    stLENS1_750[835].fEnergy := 31673.702636; stLENS1_750[835].fLow := 3.913613; stLENS1_750[835].fHigh := 9.337805; 
    stLENS1_750[836].fEnergy := 31737.113431; stLENS1_750[836].fLow := 3.899151; stLENS1_750[836].fHigh := 9.298086; 
    stLENS1_750[837].fEnergy := 31800.651174; stLENS1_750[837].fLow := 3.884743; stLENS1_750[837].fHigh := 9.258535; 
    stLENS1_750[838].fEnergy := 31864.316120; stLENS1_750[838].fLow := 3.870389; stLENS1_750[838].fHigh := 9.219153; 
    stLENS1_750[839].fEnergy := 31928.108524; stLENS1_750[839].fLow := 3.856087; stLENS1_750[839].fHigh := 9.179939; 
    stLENS1_750[840].fEnergy := 31992.028640; stLENS1_750[840].fLow := 3.841838; stLENS1_750[840].fHigh := 9.140891; 
    stLENS1_750[841].fEnergy := 32056.076724; stLENS1_750[841].fLow := 3.827642; stLENS1_750[841].fHigh := 9.102009; 
    stLENS1_750[842].fEnergy := 32120.253032; stLENS1_750[842].fLow := 3.813498; stLENS1_750[842].fHigh := 9.063293; 
    stLENS1_750[843].fEnergy := 32184.557822; stLENS1_750[843].fLow := 3.799407; stLENS1_750[843].fHigh := 9.024741; 
    stLENS1_750[844].fEnergy := 32248.991349; stLENS1_750[844].fLow := 3.785367; stLENS1_750[844].fHigh := 8.986354; 
    stLENS1_750[845].fEnergy := 32313.553873; stLENS1_750[845].fLow := 3.771380; stLENS1_750[845].fHigh := 8.948129; 
    stLENS1_750[846].fEnergy := 32378.245651; stLENS1_750[846].fLow := 3.757444; stLENS1_750[846].fHigh := 8.910067; 
    stLENS1_750[847].fEnergy := 32443.066942; stLENS1_750[847].fLow := 3.743559; stLENS1_750[847].fHigh := 8.872167; 
    stLENS1_750[848].fEnergy := 32508.018005; stLENS1_750[848].fLow := 3.729726; stLENS1_750[848].fHigh := 8.834429; 
    stLENS1_750[849].fEnergy := 32573.099101; stLENS1_750[849].fLow := 3.715944; stLENS1_750[849].fHigh := 8.796851; 
    stLENS1_750[850].fEnergy := 32638.310488; stLENS1_750[850].fLow := 3.702213; stLENS1_750[850].fHigh := 8.759432; 
    stLENS1_750[851].fEnergy := 32703.652430; stLENS1_750[851].fLow := 3.688533; stLENS1_750[851].fHigh := 8.722173; 
    stLENS1_750[852].fEnergy := 32769.125185; stLENS1_750[852].fLow := 3.674903; stLENS1_750[852].fHigh := 8.685073; 
    stLENS1_750[853].fEnergy := 32834.729018; stLENS1_750[853].fLow := 3.661324; stLENS1_750[853].fHigh := 8.648130; 
    stLENS1_750[854].fEnergy := 32900.464189; stLENS1_750[854].fLow := 3.647795; stLENS1_750[854].fHigh := 8.611344; 
    stLENS1_750[855].fEnergy := 32966.330962; stLENS1_750[855].fLow := 3.634316; stLENS1_750[855].fHigh := 8.574715; 
    stLENS1_750[856].fEnergy := 33032.329601; stLENS1_750[856].fLow := 3.620886; stLENS1_750[856].fHigh := 8.538241; 
    stLENS1_750[857].fEnergy := 33098.460369; stLENS1_750[857].fLow := 3.607507; stLENS1_750[857].fHigh := 8.501923; 
    stLENS1_750[858].fEnergy := 33164.723530; stLENS1_750[858].fLow := 3.594176; stLENS1_750[858].fHigh := 8.465759; 
    stLENS1_750[859].fEnergy := 33231.119351; stLENS1_750[859].fLow := 3.580895; stLENS1_750[859].fHigh := 8.429749; 
    stLENS1_750[860].fEnergy := 33297.648096; stLENS1_750[860].fLow := 3.567663; stLENS1_750[860].fHigh := 8.393893; 
    stLENS1_750[861].fEnergy := 33364.310032; stLENS1_750[861].fLow := 3.554480; stLENS1_750[861].fHigh := 8.358188; 
    stLENS1_750[862].fEnergy := 33431.105426; stLENS1_750[862].fLow := 3.541346; stLENS1_750[862].fHigh := 8.322636; 
    stLENS1_750[863].fEnergy := 33498.034543; stLENS1_750[863].fLow := 3.528260; stLENS1_750[863].fHigh := 8.287235; 
    stLENS1_750[864].fEnergy := 33565.097653; stLENS1_750[864].fLow := 3.515222; stLENS1_750[864].fHigh := 8.251984; 
    stLENS1_750[865].fEnergy := 33632.295023; stLENS1_750[865].fLow := 3.502233; stLENS1_750[865].fHigh := 8.216883; 
    stLENS1_750[866].fEnergy := 33699.626923; stLENS1_750[866].fLow := 3.489292; stLENS1_750[866].fHigh := 8.181932; 
    stLENS1_750[867].fEnergy := 33767.093621; stLENS1_750[867].fLow := 3.476398; stLENS1_750[867].fHigh := 8.147129; 
    stLENS1_750[868].fEnergy := 33834.695387; stLENS1_750[868].fLow := 3.463552; stLENS1_750[868].fHigh := 8.112475; 
    stLENS1_750[869].fEnergy := 33902.432493; stLENS1_750[869].fLow := 3.450754; stLENS1_750[869].fHigh := 8.077968; 
    stLENS1_750[870].fEnergy := 33970.305208; stLENS1_750[870].fLow := 3.438003; stLENS1_750[870].fHigh := 8.043607; 
    stLENS1_750[871].fEnergy := 34038.313804; stLENS1_750[871].fLow := 3.425299; stLENS1_750[871].fHigh := 8.009393; 
    stLENS1_750[872].fEnergy := 34106.458554; stLENS1_750[872].fLow := 3.412642; stLENS1_750[872].fHigh := 7.975324; 
    stLENS1_750[873].fEnergy := 34174.739729; stLENS1_750[873].fLow := 3.400032; stLENS1_750[873].fHigh := 7.941400; 
    stLENS1_750[874].fEnergy := 34243.157604; stLENS1_750[874].fLow := 3.387468; stLENS1_750[874].fHigh := 7.907621; 
    stLENS1_750[875].fEnergy := 34311.712451; stLENS1_750[875].fLow := 3.374951; stLENS1_750[875].fHigh := 7.873985; 
    stLENS1_750[876].fEnergy := 34380.404545; stLENS1_750[876].fLow := 3.362480; stLENS1_750[876].fHigh := 7.840492; 
    stLENS1_750[877].fEnergy := 34449.234161; stLENS1_750[877].fLow := 3.350055; stLENS1_750[877].fHigh := 7.807142; 
    stLENS1_750[878].fEnergy := 34518.201574; stLENS1_750[878].fLow := 3.337676; stLENS1_750[878].fHigh := 7.773933; 
    stLENS1_750[879].fEnergy := 34587.307059; stLENS1_750[879].fLow := 3.325342; stLENS1_750[879].fHigh := 7.740866; 
    stLENS1_750[880].fEnergy := 34656.550894; stLENS1_750[880].fLow := 3.313055; stLENS1_750[880].fHigh := 7.707939; 
    stLENS1_750[881].fEnergy := 34725.933355; stLENS1_750[881].fLow := 3.300813; stLENS1_750[881].fHigh := 7.675153; 
    stLENS1_750[882].fEnergy := 34795.454720; stLENS1_750[882].fLow := 3.288615; stLENS1_750[882].fHigh := 7.642506; 
    stLENS1_750[883].fEnergy := 34865.115267; stLENS1_750[883].fLow := 3.276463; stLENS1_750[883].fHigh := 7.609998; 
    stLENS1_750[884].fEnergy := 34934.915274; stLENS1_750[884].fLow := 3.264356; stLENS1_750[884].fHigh := 7.577628; 
    stLENS1_750[885].fEnergy := 35004.855021; stLENS1_750[885].fLow := 3.252294; stLENS1_750[885].fHigh := 7.545396; 
    stLENS1_750[886].fEnergy := 35074.934788; stLENS1_750[886].fLow := 3.240276; stLENS1_750[886].fHigh := 7.513300; 
    stLENS1_750[887].fEnergy := 35145.154854; stLENS1_750[887].fLow := 3.228303; stLENS1_750[887].fHigh := 7.481342; 
    stLENS1_750[888].fEnergy := 35215.515501; stLENS1_750[888].fLow := 3.216374; stLENS1_750[888].fHigh := 7.449519; 
    stLENS1_750[889].fEnergy := 35286.017010; stLENS1_750[889].fLow := 3.204489; stLENS1_750[889].fHigh := 7.417832; 
    stLENS1_750[890].fEnergy := 35356.659663; stLENS1_750[890].fLow := 3.192648; stLENS1_750[890].fHigh := 7.386279; 
    stLENS1_750[891].fEnergy := 35427.443743; stLENS1_750[891].fLow := 3.180850; stLENS1_750[891].fHigh := 7.354861; 
    stLENS1_750[892].fEnergy := 35498.369532; stLENS1_750[892].fLow := 3.169097; stLENS1_750[892].fHigh := 7.323576; 
    stLENS1_750[893].fEnergy := 35569.437315; stLENS1_750[893].fLow := 3.157386; stLENS1_750[893].fHigh := 7.292425; 
    stLENS1_750[894].fEnergy := 35640.647376; stLENS1_750[894].fLow := 3.145719; stLENS1_750[894].fHigh := 7.261406; 
    stLENS1_750[895].fEnergy := 35712.000000; stLENS1_750[895].fLow := 3.134095; stLENS1_750[895].fHigh := 7.230519; 
    stLENS1_750[896].fEnergy := 35783.495472; stLENS1_750[896].fLow := 3.122514; stLENS1_750[896].fHigh := 7.199763; 
    stLENS1_750[897].fEnergy := 35855.134077; stLENS1_750[897].fLow := 3.110976; stLENS1_750[897].fHigh := 7.169138; 
    stLENS1_750[898].fEnergy := 35926.916104; stLENS1_750[898].fLow := 3.099481; stLENS1_750[898].fHigh := 7.138643; 

    bInitialized := TRUE;
END_IF

END_FUNCTION_BLOCK

// ---- POUs/FB_LENS_SYSTEM.TcPOU
FUNCTION_BLOCK FB_LENS_SYSTEM
VAR_INPUT
    LENSES : ARRAY[1..10] OF LENS;  //Array of lens structures
    COUNT  : INT;                   //Number of lenses
    IF_NONE : LREAL := 10000.0;	    //Effective radius if no lenses are inserted (instead of infinity)
END_VAR
VAR_OUTPUT
    UNKNOWN_FAULT : BOOL;         //Fault for unknown lens state
    EFF_RADII     : REAL; //Calculated effective radii
    IN_COUNT 	  : INT;
END_VAR
VAR
    INDEX : INT;                  //Increment for loop
    KNOWN : INT;                  //Number of known lenses
    RADII : ARRAY[1..10] OF REAL; //Inserted Radii
END_VAR

(* FB_LENS_SYSTEM

Monitor an array of lens objects, updating the effective radius and positions of each.
Both the position of the lenses and the combined radius can cause a fault which is
communicated to the MPS system.

*)

//Check positions of lenses
///////////////////////////
KNOWN := 0; //Tally of known lenses
IN_COUNT := 0;

FOR INDEX := 1 TO COUNT BY 1 DO
    IF LENSES[INDEX].IN THEN
        //Inserted lenses are inserted into array
        RADII[INDEX] := LENSES[INDEX].RADIUS;
        IN_COUNT := IN_COUNT + 1;
    ELSE
        //Removed lenses are set to 0.0
        RADII[INDEX] := 0.0;
    END_IF

    // Count all known lenses
    IF LENSES[INDEX].KNOWN THEN
        KNOWN := KNOWN +1;
    END_IF
END_FOR;

// Make sure we have accounted for all lenses
UNKNOWN_FAULT := NOT (COUNT=KNOWN);

// Calculate effective radii of inserted lens
//////////////////////////////////////////////
EFF_RADII := F_EFF_RADIUS(RADII:=RADII, COUNT:=COUNT, IF_NONE:=LREAL_TO_REAL(IF_NONE));

END_FUNCTION_BLOCK

// ---- POUs/F_EFF_RADIUS.TcPOU
FUNCTION F_EFF_RADIUS : REAL
VAR_INPUT
    RADII : ARRAY[1..10] OF REAL; // Array of Effective Radii
    COUNT : INT;                 //  Number of Lenses
    IF_NONE: REAL;              //  Radius to report if none inserted (-> infinity)
END_VAR
VAR
    INDEX: INT; //Counter for Loop
END_VAR

(*F_EFF_RADIUS

Calculate the effective radius of an array of given lens radii. Non-zero elements
up to the count value are summed in reciprocal space and then inverted to give the
final calculation.
*)

// Initialize
F_EFF_RADIUS := 0.0;

//Sum Reciprocals
WHILE INDEX < COUNT+1 DO
    //Add non-zero element to total
    IF RADII[INDEX] > 0.0 THEN
        F_EFF_RADIUS := F_EFF_RADIUS + 1/RADII[INDEX];
    END_IF
    //Increment
    INDEX := INDEX + 1;
END_WHILE

//Invert if non-zero
/////////////////////
IF F_EFF_RADIUS > 0.0 THEN
    F_EFF_RADIUS := 1/F_EFF_RADIUS;
ELSE
    // B
    F_EFF_RADIUS := IF_NONE;
END_IF

END_FUNCTION

// ---- POUs/Modbus/p_ModbusTx_OutputCoils.TcPOU
PROGRAM p_ModbusTx_OutputCoils
VAR
END_VAR

mb_Output_Coils[0]:=FALSE;  //System Controls
mb_Output_Coils[1]:=FALSE;  //System Controls
mb_Output_Coils[2]:=FALSE;  //System Controls
mb_Output_Coils[3]:=FALSE;  //System Controls
mb_Output_Coils[4]:=FALSE;  //System Controls
mb_Output_Coils[5]:=FALSE;  //System Controls
mb_Output_Coils[6]:=FALSE;  //System Controls
mb_Output_Coils[7]:=FALSE;  //System Controls
mb_Output_Coils[8]:=FALSE;  //System Controls
mb_Output_Coils[9]:=FALSE;  //System Controls
mb_Output_Coils[10]:=FALSE;  //Valve switch controls
mb_Output_Coils[11]:=FALSE;  //Valve switch controls
mb_Output_Coils[12]:=FALSE;  //Valve switch controls
mb_Output_Coils[13]:=FALSE;  //Valve switch controls
mb_Output_Coils[14]:=FALSE;  //Valve switch controls
mb_Output_Coils[15]:=FALSE;  //Valve switch controls
mb_Output_Coils[16]:=FALSE;  //Valve switch controls
mb_Output_Coils[17]:=FALSE;  //Valve switch controls
mb_Output_Coils[18]:=FALSE;  //Valve switch controls
mb_Output_Coils[19]:=FALSE;  //Valve switch controls
mb_Output_Coils[20]:=FALSE;  //Valve switch controls
mb_Output_Coils[21]:=FALSE;  //Valve switch controls
mb_Output_Coils[22]:=FALSE;  //Valve switch controls
mb_Output_Coils[23]:=FALSE;  //Valve switch controls
mb_Output_Coils[24]:=FALSE;  //Valve switch controls
mb_Output_Coils[25]:=FALSE;  //Valve switch controls
mb_Output_Coils[26]:=FALSE;  //Valve switch controls
mb_Output_Coils[27]:=FALSE;  //Valve switch controls
mb_Output_Coils[28]:=FALSE;  //Valve switch controls
mb_Output_Coils[29]:=FALSE;  //Valve switch controls
mb_Output_Coils[30]:=FALSE;  //Valve switch controls
mb_Output_Coils[31]:=FALSE;  //Valve switch controls
mb_Output_Coils[32]:=FALSE;  //Valve switch controls
mb_Output_Coils[33]:=FALSE;  //Valve switch controls
mb_Output_Coils[34]:=FALSE;  //Valve switch controls
mb_Output_Coils[35]:=FALSE;  //Valve switch controls
mb_Output_Coils[36]:=FALSE;  //Valve switch controls
mb_Output_Coils[37]:=FALSE;  //Valve switch controls
mb_Output_Coils[38]:=FALSE;  //Valve switch controls
mb_Output_Coils[39]:=FALSE;  //Valve switch controls
mb_Output_Coils[40]:=FALSE;  //Valve switch controls
mb_Output_Coils[41]:=FALSE;  //Valve switch controls
mb_Output_Coils[42]:=FALSE;  //Valve switch controls
mb_Output_Coils[43]:=FALSE;  //Valve switch controls
mb_Output_Coils[44]:=FALSE;  //Valve switch controls
mb_Output_Coils[45]:=FALSE;  //Valve switch controls
mb_Output_Coils[46]:=FALSE;  //Valve switch controls
mb_Output_Coils[47]:=FALSE;  //Valve switch controls
mb_Output_Coils[48]:=FALSE;  //Valve switch controls
mb_Output_Coils[49]:=FALSE;  //Valve switch controls
mb_Output_Coils[50]:=FALSE;  //Valve switch controls
mb_Output_Coils[51]:=FALSE;  //Valve switch controls
mb_Output_Coils[52]:=FALSE;  //Valve switch controls
mb_Output_Coils[53]:=FALSE;  //Valve switch controls
mb_Output_Coils[54]:=FALSE;  //Valve switch controls
mb_Output_Coils[55]:=FALSE;  //Valve switch controls
mb_Output_Coils[56]:=FALSE;  //Valve switch controls
mb_Output_Coils[57]:=FALSE;  //Valve switch controls
mb_Output_Coils[58]:=FALSE;  //Valve switch controls
mb_Output_Coils[59]:=FALSE;  //Valve switch controls
mb_Output_Coils[60]:=FALSE;  //Valve switch controls
mb_Output_Coils[61]:=FALSE;  //Valve switch controls
mb_Output_Coils[62]:=FALSE;  //Valve switch controls
mb_Output_Coils[63]:=FALSE;  //Valve switch controls
mb_Output_Coils[64]:=FALSE;  //Valve switch controls
mb_Output_Coils[65]:=FALSE;  //Valve switch controls
mb_Output_Coils[66]:=FALSE;  //Valve switch controls
mb_Output_Coils[67]:=FALSE;  //Valve switch controls
mb_Output_Coils[68]:=FALSE;  //Valve switch controls
mb_Output_Coils[69]:=FALSE;  //Valve switch controls
mb_Output_Coils[70]:=FALSE;  //Turbo Controls
mb_Output_Coils[71]:=FALSE;  //Turbo Controls
mb_Output_Coils[72]:=FALSE;  //Turbo Controls
mb_Output_Coils[74]:=FALSE;  //Turbo Controls
mb_Output_Coils[75]:=FALSE;  //Turbo Controls
mb_Output_Coils[76]:=FALSE;  //Turbo Controls
mb_Output_Coils[77]:=FALSE;  //Turbo Controls
mb_Output_Coils[78]:=FALSE;  //Turbo Controls
mb_Output_Coils[79]:=FALSE;  //Turbo Controls
mb_Output_Coils[80]:=FALSE;  //Turbo Controls
mb_Output_Coils[81]:=FALSE;  //Turbo Controls
mb_Output_Coils[82]:=FALSE;  //Turbo Controls
mb_Output_Coils[83]:=FALSE;  //Turbo Controls
mb_Output_Coils[84]:=FALSE;  //Turbo Controls
mb_Output_Coils[85]:=FALSE;  //Turbo Controls
mb_Output_Coils[86]:=FALSE;  //Turbo Controls
mb_Output_Coils[87]:=FALSE;  //Turbo Controls
mb_Output_Coils[88]:=FALSE;  //Turbo Controls
mb_Output_Coils[89]:=FALSE;  //Turbo Controls
mb_Output_Coils[90]:=FALSE;  //Turbo Controls
mb_Output_Coils[91]:=FALSE;  //Turbo Controls
mb_Output_Coils[92]:=FALSE;  //Turbo Controls
mb_Output_Coils[93]:=FALSE;  //Turbo Controls
mb_Output_Coils[94]:=FALSE;  //Turbo Controls
mb_Output_Coils[95]:=FALSE;  //Turbo Controls
mb_Output_Coils[96]:=FALSE;  //Turbo Controls
mb_Output_Coils[97]:=FALSE;  //Turbo Controls
mb_Output_Coils[98]:=FALSE;  //Turbo Controls
mb_Output_Coils[99]:=FALSE;  //Turbo Controls
mb_Output_Coils[100]:=FALSE;  //Turbo Controls
mb_Output_Coils[101]:=FALSE;  //Turbo Controls
mb_Output_Coils[102]:=FALSE;  //Turbo Controls
mb_Output_Coils[103]:=FALSE;  //Turbo Controls
mb_Output_Coils[104]:=FALSE;  //Turbo Controls
mb_Output_Coils[105]:=FALSE;  //Turbo Controls
mb_Output_Coils[106]:=FALSE;  //Turbo Controls
mb_Output_Coils[107]:=FALSE;  //Turbo Controls
mb_Output_Coils[108]:=FALSE;  //Turbo Controls
mb_Output_Coils[109]:=FALSE;  //Turbo Controls
mb_Output_Coils[110]:=FALSE;  //Turbo Controls
mb_Output_Coils[111]:=FALSE;  //Turbo Controls
mb_Output_Coils[112]:=FALSE;  //Turbo Controls
mb_Output_Coils[113]:=FALSE;  //Turbo Controls
mb_Output_Coils[114]:=FALSE;  //Turbo Controls
mb_Output_Coils[115]:=FALSE;  //Turbo Controls
mb_Output_Coils[116]:=FALSE;  //Turbo Controls
mb_Output_Coils[117]:=FALSE;  //Turbo Controls
mb_Output_Coils[118]:=FALSE;  //Turbo Controls
mb_Output_Coils[119]:=FALSE;  //Turbo Controls
//mb_Output_Coils[120]:=vgMXT_GCC_06.xHV_SW;  //CC HV Enable
mb_Output_Coils[121]:=FALSE;  //CC HV Enable
mb_Output_Coils[122]:=FALSE;  //CC HV Enable
mb_Output_Coils[123]:=FALSE;  //CC HV Enable
mb_Output_Coils[124]:=FALSE;  //CC HV Enable
mb_Output_Coils[125]:=FALSE;  //CC HV Enable
mb_Output_Coils[126]:=FALSE;  //CC HV Enable
mb_Output_Coils[127]:=FALSE;  //CC HV Enable
mb_Output_Coils[128]:=FALSE;  //CC HV Enable
mb_Output_Coils[129]:=FALSE;  //CC HV Enable
mb_Output_Coils[130]:=FALSE;  //CC HV Enable
mb_Output_Coils[131]:=FALSE;  //CC HV Enable
mb_Output_Coils[132]:=FALSE;  //CC HV Enable
mb_Output_Coils[133]:=FALSE;  //CC HV Enable
mb_Output_Coils[134]:=FALSE;  //CC HV Enable
mb_Output_Coils[135]:=FALSE;  //CC HV Enable
mb_Output_Coils[136]:=FALSE;  //CC HV Enable
mb_Output_Coils[137]:=FALSE;  //CC HV Enable
mb_Output_Coils[138]:=FALSE;  //CC HV Enable
mb_Output_Coils[139]:=FALSE;  //CC HV Enable
mb_Output_Coils[140]:=FALSE;  //CC HV Enable
mb_Output_Coils[141]:=FALSE;  //CC HV Enable
mb_Output_Coils[142]:=FALSE;  //CC HV Enable
mb_Output_Coils[143]:=FALSE;  //CC HV Enable
mb_Output_Coils[144]:=FALSE;  //CC HV Enable
mb_Output_Coils[145]:=FALSE;  //CC HV Enable
mb_Output_Coils[146]:=FALSE;  //CC HV Enable
mb_Output_Coils[147]:=FALSE;  //CC HV Enable
mb_Output_Coils[148]:=FALSE;  //CC HV Enable
mb_Output_Coils[149]:=FALSE;  //CC HV Enable
mb_Output_Coils[150]:=FALSE;  //CC HV Enable
mb_Output_Coils[151]:=FALSE;  //CC HV Enable
mb_Output_Coils[152]:=FALSE;  //CC HV Enable
mb_Output_Coils[153]:=FALSE;  //CC HV Enable
mb_Output_Coils[154]:=FALSE;  //CC HV Enable
mb_Output_Coils[155]:=FALSE;  //CC HV Enable
mb_Output_Coils[156]:=FALSE;  //CC HV Enable
mb_Output_Coils[157]:=FALSE;  //CC HV Enable
mb_Output_Coils[158]:=FALSE;  //CC HV Enable
mb_Output_Coils[159]:=FALSE;  //CC HV Enable
mb_Output_Coils[160]:=FALSE;  //
mb_Output_Coils[161]:=FALSE;  //
mb_Output_Coils[162]:=FALSE;  //
mb_Output_Coils[163]:=FALSE;  //
mb_Output_Coils[164]:=FALSE;  //
mb_Output_Coils[165]:=FALSE;  //
mb_Output_Coils[166]:=FALSE;  //
mb_Output_Coils[167]:=FALSE;  //
mb_Output_Coils[168]:=FALSE;  //
mb_Output_Coils[169]:=FALSE;  //
mb_Output_Coils[170]:=FALSE;  //
mb_Output_Coils[171]:=FALSE;  //
mb_Output_Coils[172]:=FALSE;  //
mb_Output_Coils[173]:=FALSE;  //
mb_Output_Coils[174]:=FALSE;  //
mb_Output_Coils[175]:=FALSE;  //
mb_Output_Coils[176]:=FALSE;  //
mb_Output_Coils[177]:=FALSE;  //
mb_Output_Coils[178]:=FALSE;  //
mb_Output_Coils[179]:=FALSE;  //
mb_Output_Coils[180]:=FALSE;  //
mb_Output_Coils[181]:=FALSE;  //
mb_Output_Coils[182]:=FALSE;  //
mb_Output_Coils[183]:=FALSE;  //
mb_Output_Coils[184]:=FALSE;  //
mb_Output_Coils[185]:=FALSE;  //
mb_Output_Coils[186]:=FALSE;  //
mb_Output_Coils[187]:=FALSE;  //
mb_Output_Coils[188]:=FALSE;  //
mb_Output_Coils[189]:=FALSE;  //
mb_Output_Coils[190]:=FALSE;  //
mb_Output_Coils[191]:=FALSE;  //
mb_Output_Coils[192]:=FALSE;  //
mb_Output_Coils[193]:=FALSE;  //
mb_Output_Coils[194]:=FALSE;  //
mb_Output_Coils[195]:=FALSE;  //
mb_Output_Coils[196]:=FALSE;  //
mb_Output_Coils[197]:=FALSE;  //
mb_Output_Coils[198]:=FALSE;  //
mb_Output_Coils[199]:=FALSE;  //
mb_Output_Coils[200]:=FALSE;  //Valve overrides
mb_Output_Coils[201]:=FALSE;  //Valve overrides
mb_Output_Coils[202]:=FALSE;  //Valve overrides
mb_Output_Coils[203]:=FALSE;  //Valve overrides
mb_Output_Coils[204]:=FALSE;  //
mb_Output_Coils[205]:=FALSE;  //
mb_Output_Coils[206]:=FALSE;  //
mb_Output_Coils[207]:=FALSE;  //
mb_Output_Coils[208]:=FALSE;  //
mb_Output_Coils[209]:=FALSE;  //
mb_Output_Coils[210]:=FALSE;  //
mb_Output_Coils[211]:=FALSE;  //
mb_Output_Coils[212]:=FALSE;  //
mb_Output_Coils[213]:=FALSE;  //
mb_Output_Coils[214]:=FALSE;  //
mb_Output_Coils[215]:=FALSE;  //
mb_Output_Coils[216]:=FALSE;  //
mb_Output_Coils[217]:=FALSE;  //
mb_Output_Coils[218]:=FALSE;  //
mb_Output_Coils[219]:=FALSE;  //
mb_Output_Coils[220]:=FALSE;  //
mb_Output_Coils[221]:=FALSE;  //
mb_Output_Coils[222]:=FALSE;  //
mb_Output_Coils[223]:=FALSE;  //
mb_Output_Coils[224]:=FALSE;  //
mb_Output_Coils[225]:=FALSE;  //
mb_Output_Coils[226]:=FALSE;  //
mb_Output_Coils[227]:=FALSE;  //
mb_Output_Coils[228]:=FALSE;  //
mb_Output_Coils[229]:=FALSE;  //
mb_Output_Coils[230]:=FALSE;  //
mb_Output_Coils[231]:=FALSE;  //
mb_Output_Coils[232]:=FALSE;  //
mb_Output_Coils[233]:=FALSE;  //
mb_Output_Coils[234]:=FALSE;  //
mb_Output_Coils[235]:=FALSE;  //
mb_Output_Coils[236]:=FALSE;  //
mb_Output_Coils[237]:=FALSE;  //
mb_Output_Coils[238]:=FALSE;  //
mb_Output_Coils[239]:=FALSE;  //
mb_Output_Coils[240]:=FALSE;  //
mb_Output_Coils[241]:=FALSE;  //
mb_Output_Coils[242]:=FALSE;  //
mb_Output_Coils[243]:=FALSE;  //
mb_Output_Coils[244]:=FALSE;  //
mb_Output_Coils[245]:=FALSE;  //
mb_Output_Coils[246]:=FALSE;  //
mb_Output_Coils[247]:=FALSE;  //
mb_Output_Coils[248]:=FALSE;  //
mb_Output_Coils[249]:=FALSE;  //
mb_Output_Coils[250]:=FALSE;  //
mb_Output_Coils[251]:=FALSE;  //
mb_Output_Coils[252]:=FALSE;  //
mb_Output_Coils[253]:=FALSE;  //
mb_Output_Coils[254]:=FALSE;  //
mb_Output_Coils[255]:=FALSE;  //

END_PROGRAM
